// TwinCAT 3 PLC project GreenLine
// ProgramVersion: 3.1.4023.0
// libraries:
//   Tc2_Standard, * (Beckhoff Automation GmbH)
//   Tc2_System, * (Beckhoff Automation GmbH)
//   Tc3_Module, * (Beckhoff Automation GmbH)
// project tree:
//   GVLs/ GVL.TcGVL
//   / PlcTask.TcTTO
//   POUs/ MAIN.TcPOU
// (motion and I/O tree: see PLC project redline)
// real-time tasks:
//   TASK PlcTask: cycle T#10ms, priority 20, ADS port 350
//   TASK PlcTask1: cycle T#10ms, priority 21, ADS port 351

CONFIGURATION GreenLine
    RESOURCE PLC ON TwinCAT3
        TASK PlcTask(INTERVAL := T#10ms, PRIORITY := 21);
        PROGRAM MAIN WITH PlcTask : MAIN;
    END_RESOURCE
END_CONFIGURATION

// ---- GVLs/GVL.TcGVL
{attribute 'qualified_only'}
VAR_GLOBAL

mInSwitch : ARRAY[0..150] OF DINT;
mOutSwitch : ARRAY[0..150] OF DINT;
mInOccupancies : ARRAY[0..150] OF DINT;
mOutOccupancies : ARRAY[0..150] OF DINT;
mInSpeeds : ARRAY[0..150] OF DINT;
mOutSpeeds : ARRAY[0..150] OF DINT;
mInAuthorities : ARRAY[0..150] OF DINT;
mOutAuthorities : ARRAY[0..150] OF DINT;
mInCrossings : ARRAY[0..150] OF DINT;
mOutCrossings : ARRAY[0..150] OF DINT;
mInLeftLights : ARRAY[0..150] OF DINT;
mOutLeftLights : ARRAY[0..150] OF DINT;
mInRightLights : ARRAY[0..150] OF DINT;
mOutRightLights : ARRAY[0..150] OF DINT;
mInMaintenance : ARRAY[0..150] OF DINT;
mOutMaintenance : ARRAY[0..150] OF DINT;
mInRoute : ARRAY[0..150] OF DINT;
mOutRoute : ARRAY[0..150] OF DINT;
mSpeedLimits : ARRAY[0..150] OF DINT := [45,45,45,45,45,45,45,45,45,45,
										 45,45,70,70,70,70,60,60,60,60,
                    					 70,70,70,70,70,70,30,30,30,30,
										 30,30,30,30,30,30,30,30,30,30,
										 30,30,30,30,30,30,30,30,30,30,
										 30,30,30,30,30,30,30,30,30,30,
										 30,30,70,70,70,70,40,40,40,40,
										 40,40,40,40,40,40,70,70,70,70,
										 70,70,70,70,70,25,25,25,25,25,
										 25,25,25,25,25,25,25,25,25,25,
										 26,28,28,28,28,28,28,28,28,30,
										 30,30,30,30,30,30,15,15,15,15,
										 15,20,20,20,20,20,20,20,20,20,
										 20,20,20,20,20,20,20,20,20,20,
										 20,20,20,20,20,20,20,20,20,20,100];

END_VAR

// ---- POUs/MAIN.TcPOU
PROGRAM MAIN
VAR

inc1 : DINT := 0;

END_VAR

FOR inc1 := 0 TO 150 DO
	//Sets Red Lights
	IF GVL.mInOccupancies[inc1] = 0
	THEN
		GVL.mOutLeftLights[inc1] := 0;
		GVL.mOutRightLights[inc1] := 0;
	//Sets green lights
	ELSE
		GVL.mOutLeftLights[inc1] := 2;
		GVL.mOutRightLights[inc1] := 2;
	END_IF
END_FOR

FOR inc1 := 1 TO 149 DO
	//Sets Yellow Lights
	IF GVL.mInOccupancies[inc1-1] = 0 AND GVL.mInOccupancies[inc1] <> 0
	THEN
		GVL.mOutRightLights[inc1] := 1;
	END_IF
	IF GVL.mInOccupancies[inc1+1] = 0 AND GVL.mInOccupancies[inc1] <> 0
	THEN
	GVL.mOutLeftLights[inc1] := 1;
	END_IF
END_FOR

//0 to 61 corresponds to blocks 1 to 62
//76 to 150 corresponds to 

FOR inc1 := 0 TO 150 DO

	GVL.mOutOccupancies[inc1] := GVL.mInOccupancies[inc1];
	GVL.mOutSpeeds[inc1] := GVL.mInSpeeds[inc1];
	GVL.mOutAuthorities[inc1] := GVL.mInAuthorities[inc1];
	GVL.mOutMaintenance[inc1] := GVL.mInMaintenance[inc1];
	IF GVL.mInSpeeds[inc1] < GVL.mSpeedLimits[inc1]
	THEN
		GVL.mOutSpeeds[inc1] := GVL.mInSpeeds[inc1];
	ELSE
		GVL.mOutSpeeds[inc1] := GVL.mSpeedLimits[inc1];
	END_IF

END_FOR

inc1 := 0;

//This starts the main track logic section

//Crossing Logic
IF GVL.mInOccupancies[18] = 0 THEN
	GVL.mOutCrossings[18] := 1;
ELSE
	GVL.mOutCrossings[18] := 0;
END_IF


//Switch Logic

//Set switch on block 13
IF GVL.mInMaintenance[12] = 1 THEN
    GVL.mOutSwitch[12] := GVL.mInSwitch[12];
ELSE
    IF GVL.mInOccupancies[11] = 0 THEN
    	GVL.mOutSwitch[12] := 11;
    ELSE
		GVL.mOutSwitch[12] := 0;
	END_IF
END_IF

//Set switch on block 29
IF GVL.mInMaintenance[28] = 1 THEN
    GVL.mOutSwitch[28] := GVL.mInSwitch[28];
ELSE
    IF GVL.mInOccupancies[28] = 0 THEN
    FOR inc1 := 12 TO 28 DO 
        IF GVL.mInOccupancies[inc1] = 0 THEN
            GVL.mOutSwitch[28] := 149;
            Exit;
        ELSE 
            GVL.mOutSwitch[28] := 29;
        END_IF
    END_FOR
	END_IF
END_IF


//Set switch on block 58
IF GVL.mInMaintenance[57] = 1 THEN
    GVL.mOutSwitch[57] := GVL.mInSwitch[57];
ELSE
	GVL.mOutSwitch[57] := 58;
END_IF
	
//Set switch on block
IF GVL.mInMaintenance[76] = 1 THEN
    GVL.mOutSwitch[76] := GVL.mInSwitch[76];
ELSE
    IF GVL.mInOccupancies[75] = 0 THEN
    FOR inc1 := 76 TO 84 DO 
        IF GVL.mInOccupancies[inc1] = 0 THEN
            GVL.mOutSwitch[75] := 100;
            Exit;
        ELSE 
            GVL.mOutSwitch[75] := 74;
        END_IF
    END_FOR
	END_IF
END_IF

IF GVL.mInMaintenance[84] = 1 THEN
    GVL.mOutSwitch[84] := GVL.mInSwitch[84];
ELSE
    IF GVL.mInOccupancies[99] = 0 THEN
    FOR inc1 := 76 TO 84 DO 
        IF GVL.mInOccupancies[inc1] = 0 THEN
            GVL.mOutSwitch[84] := 85;
            Exit;
        ELSE 
            GVL.mOutSwitch[84] := 99;
        END_IF
    END_FOR
	END_IF
END_IF

END_PROGRAM
